PROGRAM POU_GatewaySignals
VAR
END_VAR

// NETWORK 1

END_PROGRAM

(* stored: Version 1.1.0.1, ProductVersion 3.1.4024.0
   POU POU_GatewaySignals: Id {0c5be854-7e49-473e-9daf-42593f713bc9}, SpecialFunc None *)
